{attribute 'GeneratedUsingTerminal: ELX4181-0000-0016'}
{attribute addProperty BoxType "ELX4181-0000-0016"}
{attribute addProperty Id "Ch_1Ch_1_8C75A2992WcStateAT %I*WcState_0B2B16F91InfoDataAT %I*InfoData_90184F0C16"}
{attribute addProperty CRC "1883363515"}
{attribute addProperty Size "19"}
TYPE ELX4181_7041D8BB EXTENDS EtcSlaveTerminalBase_947E5A46 :
STRUCT
	{attribute addProperty Name "Ch_1"}
	Ch_1 : Ch_1_8C75A299;
	{attribute addProperty Name "WcState"}
	WcState : WcState_0B2B16F9;
	{attribute addProperty Name "InfoData"}
	InfoData : InfoData_90184F0C;
END_STRUCT
END_TYPE

(* stored: Version 1.2.0.0, ProductVersion 3.1.4024.9
   DUT ELX4181_7041D8BB: Id {65699f92-f83b-4ec8-83cd-a892561ad798} *)
